Staubli VAL3: onF6Event.pgx

program onF6Event()
  local bool l_bStatus
begin
  // look if the bButton is enable
  if bButton[5]
  endIf
end
